Staubli VAL3: EditPath.pgx

program EditPath()
  local num l_nKey
begin
  //
  nPage=1
  bUserRefresh=bListRefresh=true
  do
    call Refresh()
    call RefreshList()
    call user:setList("路径",sList,bUserRefresh,bListRefresh,nSelected,sItem,l_nKey)
    bUserRefresh=false
    bListRefresh=false
    call MainKey(l_nKey)
    delay(0)
  until bExit
  nPage=0
  bUserRefresh=bListRefresh=true
  bExit=false
end
